PROGRAM Bootup_Shutdown_ctrl
VAR
	bIpcInput_on: BOOL;
	bXmlReadEn: BOOL;
	bCSVReadEn: BOOL;
	bCsvReadDone: BOOL;
	
	bIPCInputOnRE	: R_trig;
	bIPCOnRE		: R_Trig;
	bXmlCsvReadDoneRE : R_Trig;
	bXmlCsvWriteDoneRE	:R_trig;
	
	bCsvWriteEn: BOOL;
	bIpcOnHR: BOOL;


	
	bSFQTest: BOOL;
	bSFQTest_read: BOOL;
	

	bBootUpReadXMLDone	:BOOL;
	bShutdownWriteXMLDone	:BOOL;
	sStatus: STRING;
	bsyed: BOOL;
	bIpcOffDelay: BOOL;
	tIpcOffDelay: TON;
	test: Bool;
	
	
	
	
	
	
	
	

	
	
	
	
	bSHutdownTest: BOOL;
	
	on: BOOL;


END_VAR

VAR PERSISTENT
	bBootupHold: BOOL;
END_VAR


// IPC OFF Selector Switch - OFF
bIPCInputOnRE(CLK:=ARbDI[eX11111_IpcDcOnSignal] OR bBatteryModeActivated OR bSFQTest , Q=> );

IF ARbDI[eX11111_IpcDcOnSignal] THEN
	on:= FALSE;
	ELSE
	on:= TRUE;
	
END_IF


// IPC autoboot start signal
bIPCOnRE(CLK:=TRUE OR bSFQTest_read  , Q=> );

//IPC On Holding relay -output
IF PowerOnDelay.Q AND NOT tIpcOffDelay.Q THEN
	bIpcOnHR := TRUE;
	ELSE
	bIpcOnHR := FALSE;
END_IF

ARwDO[eY11007_IpcDcOnHoldingRelay].00:=bIpcOnHR OR bsyed;

// Bootup
IF bIPCOnRE.Q AND NOT bBootupHold THEN
	bMainCtrl:=FALSE;
	bReadXmlEn:= TRUE;
END_IF

bXmlCsvReadDoneRE(CLK:= bReadXmlComplete (*AND NOT Alarm_XMLReadnWrite.fbXmlSrvReadFromXML.bBusy AND bCsvReadDone*) , Q=> );

IF bXmlCsvReadDoneRE.Q THEN 
	bMainCtrl:=TRUE;
	bBootupHold:= TRUE;
END_IF

// Shutdown
IF bIPCInputOnRE.Q OR bSHutdownTest THEN
	bBootupHold:= FALSE;
	bMachineShutdown:=TRUE;
	bShutdownPopupPage:=TRUE;
	bRecipeShutdownRequestFlag:= TRUE;
	bCsvShutdownRequestFlag:=TRUE;
	bWriteXmlEn:= TRUE;
END_IF

bXmlCsvWriteDoneRE(CLK:= bWrite_Done (*AND bRecipeReadyToShutdownFlag AND bCsvReadyToShutdownFlag*), Q=> );

IF bXmlCsvWriteDoneRE.Q THEN
	bIpcOffDelay:= TRUE;
	bWriteXmlEn:=FALSE;
	
END_IF

tIpcOffDelay(IN:=bIpcOffDelay , PT:= T#2S , Q=> , ET=> );

END_PROGRAM

(* stored: Version 1.1.0.1, ProductVersion 3.1.4024.12
   POU Bootup_Shutdown_ctrl: Id {76222284-52aa-4a70-a63f-a16a53caa269}, SpecialFunc None *)
